FUNCTION_BLOCK PUBLIC ManualControl
VAR_INPUT
	Switch: BOOL;
END_VAR
VAR
	ManualControl: BOOL;
	TimeForInterlockDelay: TIME := T#0.05S;
	ManualMode: BOOL;
	MotorSelection_1: MotorSelection;
	SelectedMotor: INT;
	temp: TIME;
	LowerLeftInterlock: TOF;
	LowerLeft: BOOL;
	LowerRightInterlock: TOF;
	LowerRight: BOOL;
END_VAR
VAR_OUTPUT
	Output: BOOL;
END_VAR
VAR // added by the converter: edge detectors and wires of the graphical bodies
    _w1, _w2, _w3, _w4, _w5, _w6, _w7, _w8, _w9, _w10, _w11, _w12 : BOOL;
    _rt1, _rt2, _rt3, _rt4 : R_TRIG;
    _ft1, _ft2, _ft3, _ft4 : F_TRIG;
END_VAR

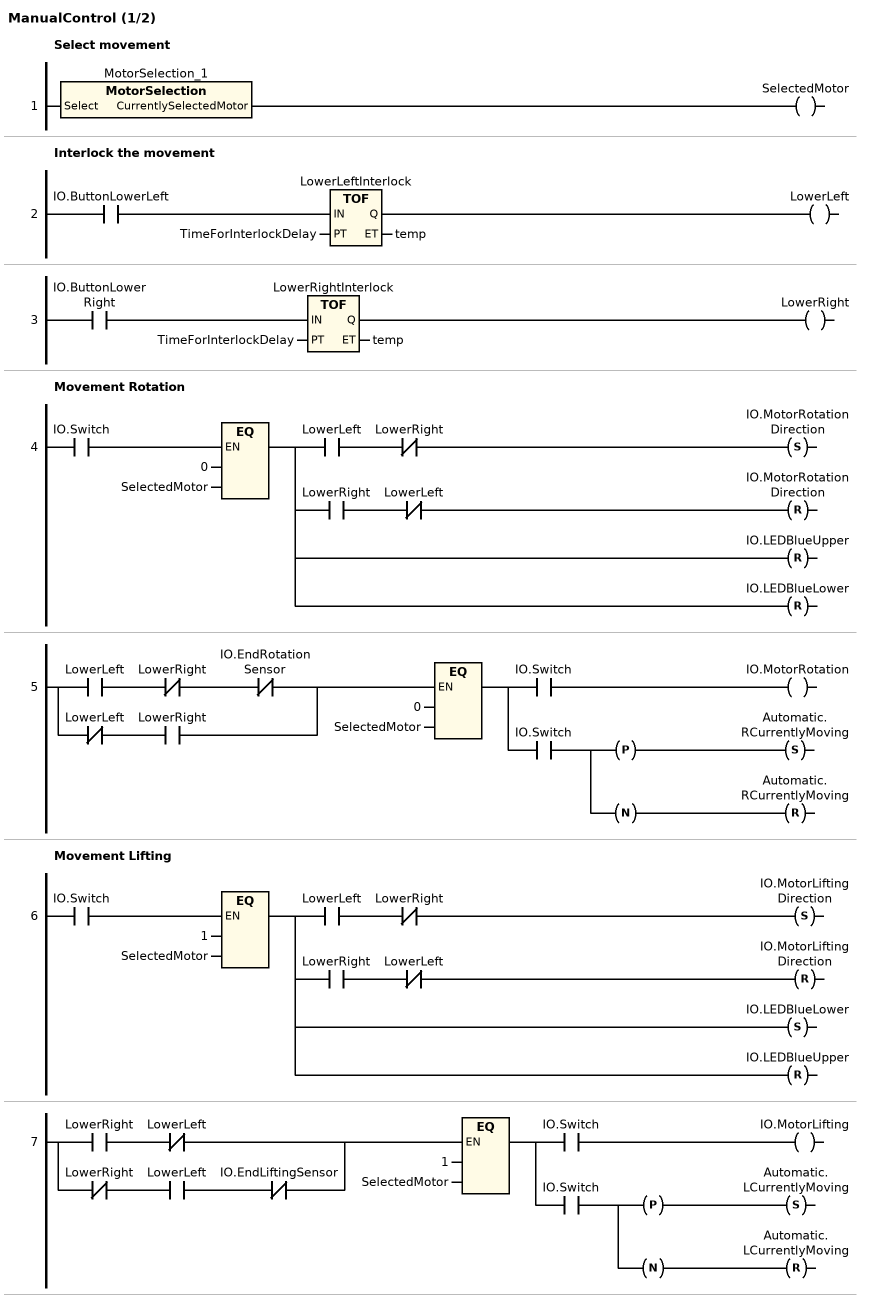
// NETWORK 1: Select movement
MotorSelection_1(Select := TRUE); // MotorSelection
SelectedMotor := MotorSelection_1.CurrentlySelectedMotor;

// NETWORK 2: Interlock the movement
LowerLeftInterlock(IN := IO.ButtonLowerLeft, PT := TimeForInterlockDelay, ET => temp); // TOF
LowerLeft := LowerLeftInterlock.Q;

// NETWORK 3
LowerRightInterlock(IN := IO.ButtonLowerRight, PT := TimeForInterlockDelay, ET => temp); // TOF
LowerRight := LowerRightInterlock.Q;

// NETWORK 4: Movement Rotation
_w1 := IO.Switch AND 0 = SelectedMotor;
IO.MotorRotationDirection S= _w1 AND LowerLeft AND NOT LowerRight;
IO.MotorRotationDirection R= _w1 AND LowerRight AND NOT LowerLeft;
IO.LEDBlueUpper R= _w1;
IO.LEDBlueLower R= _w1;

// NETWORK 5
_w2 := (LowerLeft AND NOT LowerRight AND NOT IO.EndRotationSensor OR NOT LowerLeft AND LowerRight) AND 0 = SelectedMotor;
IO.MotorRotation := _w2 AND IO.Switch;
_w3 := _w2 AND IO.Switch;
_rt1(CLK := _w3);
Automatic.RCurrentlyMoving S= _rt1.Q;
_ft1(CLK := _w3);
Automatic.RCurrentlyMoving R= _ft1.Q;

// NETWORK 6: Movement Lifting
_w4 := IO.Switch AND 1 = SelectedMotor;
IO.MotorLiftingDirection S= _w4 AND LowerLeft AND NOT LowerRight;
IO.MotorLiftingDirection R= _w4 AND LowerRight AND NOT LowerLeft;
IO.LEDBlueLower S= _w4;
IO.LEDBlueUpper R= _w4;

// NETWORK 7
_w5 := (LowerRight AND NOT LowerLeft OR NOT LowerRight AND LowerLeft AND NOT IO.EndLiftingSensor) AND 1 = SelectedMotor;
IO.MotorLifting := _w5 AND IO.Switch;
_w6 := _w5 AND IO.Switch;
_rt2(CLK := _w6);
Automatic.LCurrentlyMoving S= _rt2.Q;
_ft2(CLK := _w6);
Automatic.LCurrentlyMoving R= _ft2.Q;

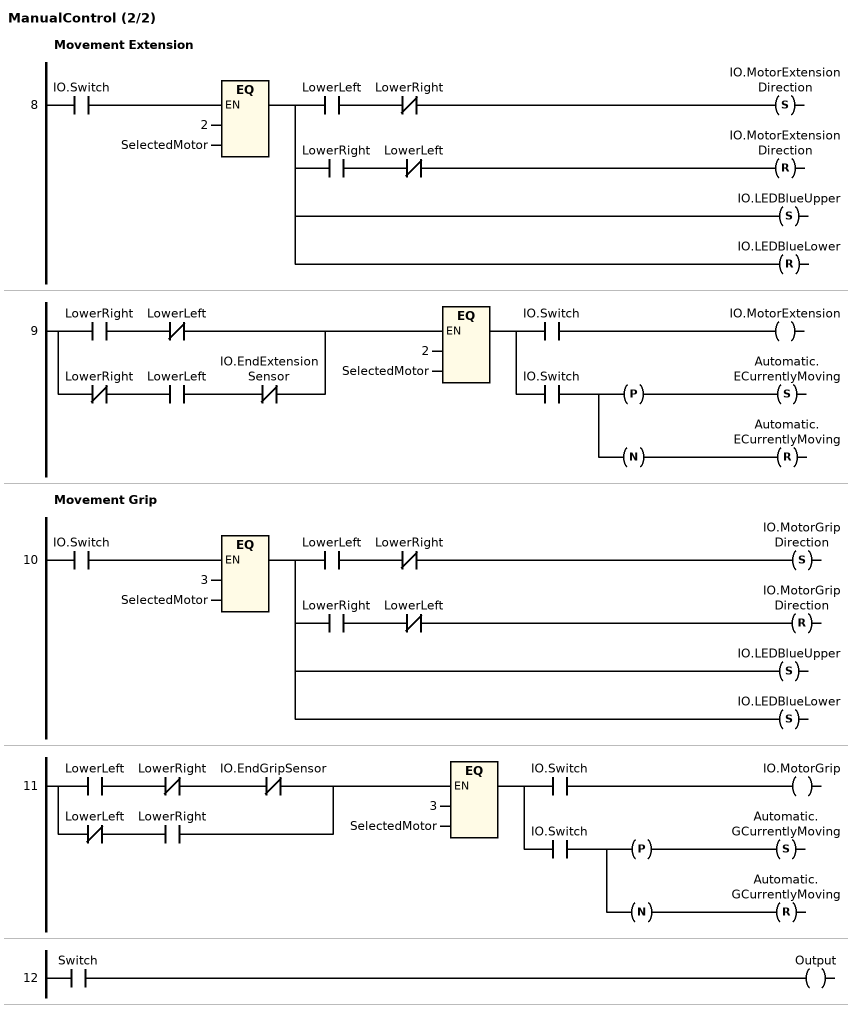
// NETWORK 8: Movement Extension
_w7 := IO.Switch AND 2 = SelectedMotor;
IO.MotorExtensionDirection S= _w7 AND LowerLeft AND NOT LowerRight;
IO.MotorExtensionDirection R= _w7 AND LowerRight AND NOT LowerLeft;
IO.LEDBlueUpper S= _w7;
IO.LEDBlueLower R= _w7;

// NETWORK 9
_w8 := (LowerRight AND NOT LowerLeft OR NOT LowerRight AND LowerLeft AND NOT IO.EndExtensionSensor) AND 2 = SelectedMotor;
IO.MotorExtension := _w8 AND IO.Switch;
_w9 := _w8 AND IO.Switch;
_rt3(CLK := _w9);
Automatic.ECurrentlyMoving S= _rt3.Q;
_ft3(CLK := _w9);
Automatic.ECurrentlyMoving R= _ft3.Q;

// NETWORK 10: Movement Grip
_w10 := IO.Switch AND 3 = SelectedMotor;
IO.MotorGripDirection S= _w10 AND LowerLeft AND NOT LowerRight;
IO.MotorGripDirection R= _w10 AND LowerRight AND NOT LowerLeft;
IO.LEDBlueUpper S= _w10;
IO.LEDBlueLower S= _w10;

// NETWORK 11
_w11 := (LowerLeft AND NOT LowerRight AND NOT IO.EndGripSensor OR NOT LowerLeft AND LowerRight) AND 3 = SelectedMotor;
IO.MotorGrip := _w11 AND IO.Switch;
_w12 := _w11 AND IO.Switch;
_rt4(CLK := _w12);
Automatic.GCurrentlyMoving S= _rt4.Q;
_ft4(CLK := _w12);
Automatic.GCurrentlyMoving R= _ft4.Q;

// NETWORK 12
Output := Switch;

END_FUNCTION_BLOCK

(* stored: Version 1.1.0.1, ProductVersion 3.1.4024.13
   POU ManualControl: Id {0dc011e3-56d5-4b91-a8d5-8c19aa1fc8c8}, SpecialFunc None *)
